PROGRAM Drad_External
VAR
    fEncoderPosition : LREAL;
    EncoderPosition AT %Q* : DINT; //Encoder value for NC
    fScaler : LREAL := 1000000;
END_VAR

astAxes[AXIS_DRAD_EXTERNAL].stInputs.bLimitBwd := TRUE;
astAxes[AXIS_DRAD_EXTERNAL].stInputs.bLimitFwd := TRUE;
astAxes[AXIS_DRAD_EXTERNAL].stControl.bEnable := TRUE;

//B = A-E
fEncoderPosition := astAxes[AXIS_DRAD].stStatus.fActPosition - astAxes[AXIS_DRAD_INTERNAL].stStatus.fActPosition;
EncoderPosition:= LREAL_TO_DINT(fEncoderPosition * fScaler);

END_PROGRAM

(* stored: Version 1.1.0.1, ProductVersion 3.1.4024.11
   POU Drad_External: Id {d9a877bc-3d1a-4d88-aa1a-28b6e1cdd406}, SpecialFunc None *)
